// Mitsubishi GX Works2 project: resist   PLC: Q03UDV

PROGRAM MAIN
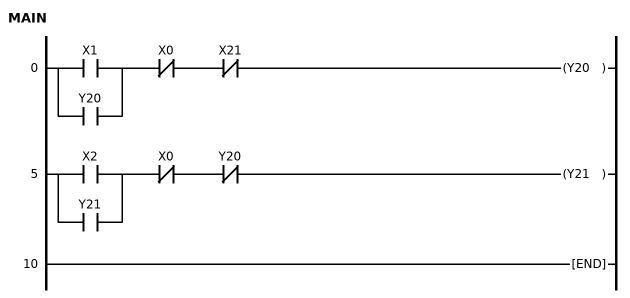
0     LD      X1
      OR      Y20
      ANI     X0
      ANI     X21
      OUT     Y20
5     LD      X2
      OR      Y21
      ANI     X0
      ANI     Y20
      OUT     Y21
10    END
END_PROGRAM
